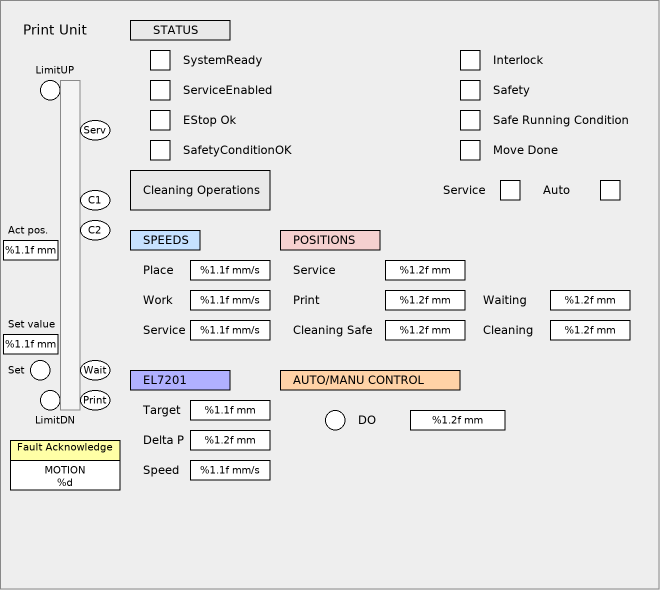
VISUALIZATION _VISU_CleanPU  // 660x590
VAR_IN_OUT
  mInst  : FB_CleaningMotorAxisPU;
END_VAR
    Rectangle (0,0 660x590)
    Polyline (200,380)
    Polyline (130,240)
    Rectangle (130,170 140x40)
    Rectangle (130,370 100x20)
    Rectangle (280,370 180x20)
    Rectangle (280,230 100x20)
    Rectangle (130,230 70x20)
    Rectangle (130,20 100x20)
    Rectangle (20,20 100x20), "Print Unit"
    Polyline (130,30)
    Polyline (230,30)
    Rectangle (150,20 60x20), "STATUS"
    RoundedRectangle (150,80 20x20), colour toggle: mInst.bI_UsrService
    RoundedRectangle (150,110 20x20), colour toggle: NOT mInst.bI_Emergency
    RoundedRectangle (150,140 20x20), colour toggle: mInst.bI_SafetyOk
    RoundedRectangle (460,140 20x20), colour toggle: NOT mInst.bL_Busy
    RoundedRectangle (150,50 20x20), colour toggle: mInst.bI_MachineReady
    Rectangle (180,50 120x20), "SystemReady"
    Rectangle (180,80 120x20), "ServiceEnabled"
    Rectangle (180,110 120x20), "EStop Ok"
    Rectangle (180,140 120x20), "SafetyConditionOK"
    Rectangle (490,140 90x20), "Move Done"
    Rectangle (290,370 170x20), "AUTO/MANU CONTROL"
    Polyline (450,380)
    Rectangle (30,60 50x20), "LimitUP"
    Ellipse (40,80 20x20), colour toggle: NOT mInst.bI_SensorTop
    Ellipse (40,390 20x20), colour toggle: NOT mInst.bI_SensorBottom
    Rectangle (30,410 50x20), "LimitDN"
    Scrollbar (60,80 20x330)
        p2245068023: 0.5
        p1057716461: mInst.fB_Axis.fO_ActualPosition
    Rectangle (140,230 70x20), "SPEEDS"
    Rectangle (190,260 80x20), "%1.1f mm/s", text variable: mInst.sI_SpeedDef.fP_PlaceSpeed
        OnMouseDown: write the text variable via VisuDialogs.Numpad
    Rectangle (190,290 80x20), "%1.1f mm/s", text variable: mInst.sI_SpeedDef.fP_WorkSpeed
        OnMouseDown: write the text variable via VisuDialogs.Numpad
    Rectangle (190,320 80x20), "%1.1f mm/s", text variable: mInst.sI_SpeedDef.fP_ServiceSpeed
        OnMouseDown: write the text variable via VisuDialogs.Numpad
    Rectangle (140,260 45x20), "Place"
    Rectangle (140,290 45x20), "Work"
    Rectangle (140,320 45x20), "Service"
        OnMouseDown: write the text variable via Edit
    Rectangle (290,260 90x20), "Service"
    Rectangle (290,290 90x20), "Print"
    Polyline (350,240)
    Rectangle (290,230 90x20), "POSITIONS"
    Rectangle (190,400 80x20), "%1.1f mm", text variable: 1000 * mInst.fB_Axis.fI_TargetPosition
    RoundedRectangle (460,80 20x20), colour toggle: mInst.bI_SafeToMove
    Rectangle (490,80 120x20), "Safety"
    RoundedRectangle (460,50 20x20), colour toggle: mInst.bI_SafeToMove
    Rectangle (490,50 120x20), "Interlock"
    Rectangle (5,360 25x20), "Set"
    Ellipse (30,360 20x20), colour toggle: mInst.fB_Axis.bI_SetPosition
        toggle mInst.fB_Axis.bI_SetPosition
    Rectangle (3,240 55x20), "%1.1f mm", text variable: 1000 * mInst.fB_Axis.fO_ActualPosition
    Rectangle (290,320 90x20), "Cleaning Safe"
    Rectangle (385,320 80x20), "%1.2f mm", text variable: mInst.fI_PositionClean1
        OnMouseDown: write the text variable via VisuDialogs.Numpad
    Rectangle (140,400 45x20), "Target"
    Rectangle (140,460 45x20), "Speed"
    Rectangle (190,460 80x20), "%1.1f mm/s", text variable: 1000 * mInst.fB_Axis.fI_SpeedLimit
    Rectangle (140,370 90x20), "EL7201"
    Rectangle (140,430 45x20), "Delta P"
    Rectangle (190,430 80x20), "%1.2f mm", text variable: 1000 * mInst.fB_Axis.fL_Delta_P
    Ellipse (80,120 30x20), "Serv", colour toggle: mInst.pInPosService
    Ellipse (80,220 30x20), "C2", colour toggle: mInst.pInPosClean2
    Ellipse (80,190 30x20), "C1", colour toggle: mInst.pInPosClean1
    Ellipse (80,360 30x20), "Wait", colour toggle: mInst.pInPosWait
    Ellipse (80,390 30x20), "Print", colour toggle: mInst.pInPosPrint
    Polyline (640,160)
    Rectangle (140,180 140x20), "Cleaning Operations"
    Polyline (270,200)
    RoundedRectangle (460,110 20x20), colour toggle: mInst.bL_SafeRunningCondition
    Rectangle (490,110 140x20), "Safe Running Condition"
    RoundedRectangle (600,180 20x20), colour toggle: mInst.bI_UsrAutoMode
    Rectangle (540,180 55x20), "Auto"
    Polyline (340,80)
    Rectangle (10,440 110x50), "Fault Acknowledge", colour toggle: (mInst.wL_ErrorCode) <> 0
    RoundedRectangle (10,460 110x30), "%d", text variable: mInst.wL_ErrorCode
        tap mInst.sADS_CleanAxis.bI_FaultAck
    RoundedRectangle (10,460 110x20), "MOTION"
    Rectangle (3,334 55x20), "%1.1f mm", text variable: mInst.fL_SetPositionValue
        OnMouseDown: write the text variable via VisuDialogs.Numpad
    Rectangle (480,320 65x20), "Cleaning"
    Rectangle (550,320 80x20), "%1.2f mm", text variable: mInst.fI_PositionClean2
        OnMouseDown: write the text variable via VisuDialogs.Numpad
    RoundedRectangle (500,180 20x20), colour toggle: mInst.bI_UsrService
    Rectangle (440,180 55x20), "Service"
    Rectangle (410,410 95x20), "%1.2f mm", text variable: mInst.sADS_CleanAxis.fI_ManualTargetPos
        OnMouseDown: write the text variable via VisuDialogs.Numpad, min mInst.sADS_CleanAxis.sO_AxisPosition.fC_Min, max mInst.sADS_CleanAxis.sO_AxisPosition.fC_Max
    Rectangle (355,410 50x20), "DO"
    Ellipse (325,410 20x20), colour toggle: mInst.sADS_CleanAxis.bI_ManualMove, input disabled if: NOT mInst.sADS_CleanAxis.bO_ManualMoveCanEx
        toggle mInst.sADS_CleanAxis.bI_ManualMove
    Rectangle (385,260 80x20), "%1.2f mm", text variable: mInst.fI_PositionService
        OnMouseDown: write the text variable via VisuDialogs.Numpad
    Rectangle (385,290 80x20), "%1.2f mm", text variable: mInst.fL_PrintPositionMM
        OnMouseDown: write the text variable via VisuDialogs.Numpad, min 0.8, max 2.5
    Rectangle (480,290 65x20), "Waiting"
    Rectangle (550,290 80x20), "%1.2f mm", text variable: mInst.fI_PositionWait
        OnMouseDown: write the text variable via VisuDialogs.Numpad
    Rectangle (5,314 50x20), "Set value"
    Rectangle (5,220 50x20), "Act pos."
END_VISUALIZATION

(* stored: Version 1.1.0.1, ProductVersion 3.1.4024.11
   Visu _VISU_CleanPU: Id {93aa0320-6bcf-4873-b800-a02f82dc1748} *)
